(* PLC project Astro, Actility iec61131 1.0.28, author Laurent Nicq *)
(* stored: creationDateTime 2013-03-20T17:09:43, version 1.1.2, modificationDateTime 2013-07-26T10:44:38 *)

(* Example for using the Sunset *)
PROGRAM POU_Astro_Using
  VAR_EXTERNAL
    GL_Astro_Status : DINT;
    GL_Current_DateTime : DT;
    GL_SunSet_Time : DT;
  END_VAR
  VAR
    Information : STRING;
    astro_status : DINT := 0;
    delay_before : TIME := t#30s;
    time_remaining : TIME;  (* temporary for debug *)
    delay_after : TIME := t#45s;
    light : BOOL := FALSE;
    current_day : DINT;
  END_VAR

(* transition new_day *)
yday(GL_Current_DateTime)<> current_day;
/* check for a different day. Avoid dealing with 365-366 days case */
              
(* Need to wait for a new day before using a
SunSet value calculated by the Astro script *)
INITIAL_STEP Get_status:
  GET_STATUS_INLINE1(N);
END_STEP
ACTION GET_STATUS_INLINE1:
  astro_status:= GL_Astro_Status;
END_ACTION
TRANSITION FROM Get_status TO Display_Status
  := astro_status <>0;
END_TRANSITION
TRANSITION FROM Get_status TO Astro_OK
  := astro_status = 0;
END_TRANSITION
STEP Display_Status:
  DISPLAY_STATUS_INLINE2(P);
END_STEP
ACTION DISPLAY_STATUS_INLINE2:
  Information:='Astro is NOT RUNNING';
END_ACTION
TRANSITION FROM Display_Status TO Get_status
  := TRUE;
END_TRANSITION
STEP Astro_OK:
  ASTRO_OK_INLINE3(P);
  store_current_day(N);
  remaining(N);
END_STEP
ACTION ASTRO_OK_INLINE3:
  Information:='Astro is RUNNING';
END_ACTION
TRANSITION FROM Astro_OK TO Start_SunSet
  := GL_Current_DateTime > GL_SunSet_Time - delay_before;
END_TRANSITION
STEP Start_SunSet:
  START_SUNSET_INLINE4(P);
END_STEP
ACTION START_SUNSET_INLINE4:
  light:=TRUE;
END_ACTION
TRANSITION FROM Start_SunSet TO Stop_SunSet
  := GL_Current_DateTime > (( GL_SunSet_Time - delay_before) + delay_after);
END_TRANSITION
STEP Stop_SunSet:
  STOP_SUNSET_INLINE5(P);
END_STEP
ACTION STOP_SUNSET_INLINE5:
  light:=FALSE;
END_ACTION
TRANSITION FROM Stop_SunSet TO Get_status
  := new_day;
END_TRANSITION

ACTION store_current_day:
current_day:= yday(GL_Current_DateTime);
              
END_ACTION

ACTION remaining:
time_remaining:= SUB_DT_DT(GL_SunSet_Time , GL_Current_DateTime);
              
END_ACTION
END_PROGRAM

(* Distributes the Sunset Sunrise times *)
PROGRAM POU_Astro_Sun_Time
  VAR_EXTERNAL
    GL_SunSet_Time : DT;
    GL_SunRise_Time : DT;
    GL_Current_DateTime : DT;
    GL_Astro_Status : INT;
    GL_Lat : REAL;
    GL_Lon : REAL;
  END_VAR
  VAR
    Astro_Version : STRING := '1.1.2';
    current_day : DINT;
    Lat : REAL := 0;
    Lon : REAL := 0;
  END_VAR

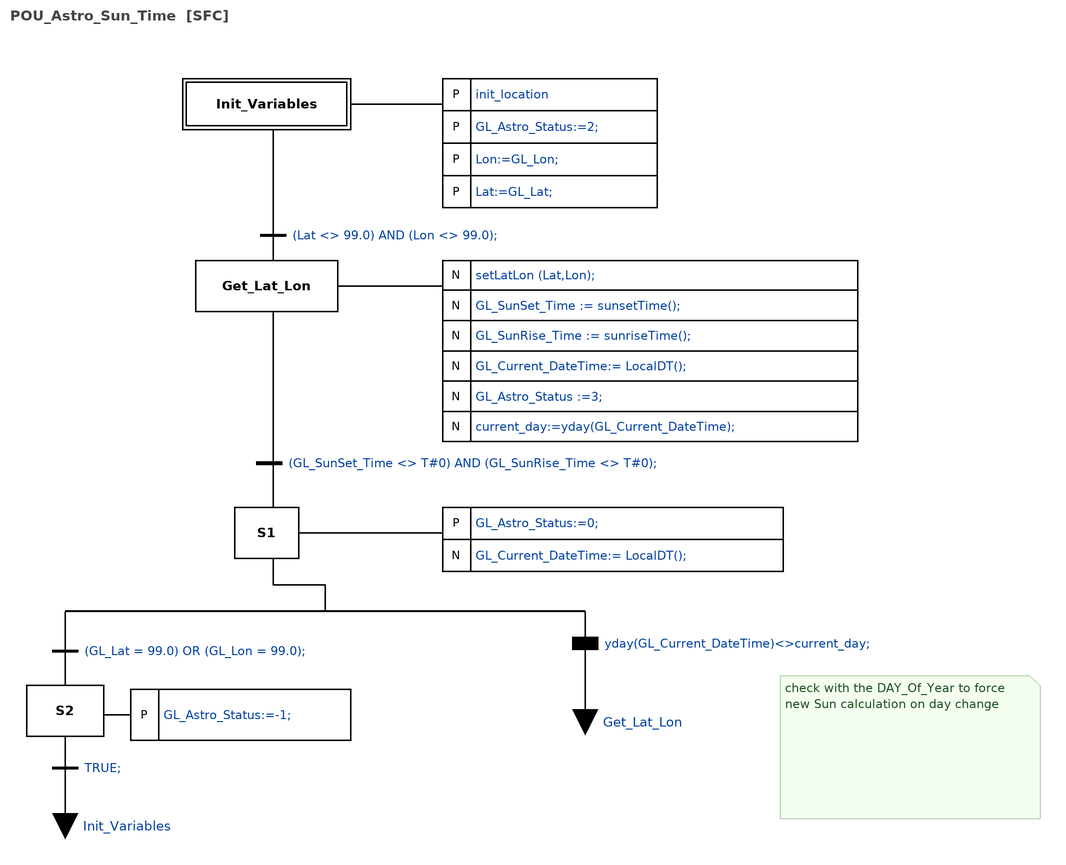
(* check with the DAY_Of_Year to force new Sun calculation on day change *)
INITIAL_STEP Init_Variables:
  init_location(P);
  INIT_VARIABLES_INLINE1(P);
  INIT_VARIABLES_INLINE2(P);
  INIT_VARIABLES_INLINE3(P);
END_STEP
ACTION INIT_VARIABLES_INLINE1:
  GL_Astro_Status:=2;
END_ACTION
ACTION INIT_VARIABLES_INLINE2:
  Lon:=GL_Lon;
END_ACTION
ACTION INIT_VARIABLES_INLINE3:
  Lat:=GL_Lat;
END_ACTION
TRANSITION FROM Init_Variables TO Get_Lat_Lon
  := (Lat <> 99.0) AND (Lon <> 99.0);
END_TRANSITION
STEP Get_Lat_Lon:
  GET_LAT_LON_INLINE4(N);
  GET_LAT_LON_INLINE5(N);
  GET_LAT_LON_INLINE6(N);
  GET_LAT_LON_INLINE7(N);
  GET_LAT_LON_INLINE8(N);
  GET_LAT_LON_INLINE9(N);
END_STEP
ACTION GET_LAT_LON_INLINE4:
  setLatLon (Lat,Lon);
END_ACTION
ACTION GET_LAT_LON_INLINE5:
  GL_SunSet_Time := sunsetTime();
END_ACTION
ACTION GET_LAT_LON_INLINE6:
  GL_SunRise_Time := sunriseTime();
END_ACTION
ACTION GET_LAT_LON_INLINE7:
  GL_Current_DateTime:= LocalDT();
END_ACTION
ACTION GET_LAT_LON_INLINE8:
  GL_Astro_Status :=3;
END_ACTION
ACTION GET_LAT_LON_INLINE9:
  current_day:=yday(GL_Current_DateTime);
END_ACTION
TRANSITION FROM Get_Lat_Lon TO S1
  := (GL_SunSet_Time <> T#0) AND (GL_SunRise_Time <> T#0);
END_TRANSITION
STEP S1:
  S1_INLINE10(P);
  S1_INLINE11(N);
END_STEP
ACTION S1_INLINE10:
  GL_Astro_Status:=0;
END_ACTION
ACTION S1_INLINE11:
  GL_Current_DateTime:= LocalDT();
END_ACTION
TRANSITION FROM S1 TO S2
  := (GL_Lat = 99.0) OR (GL_Lon = 99.0);
END_TRANSITION
TRANSITION FROM S1 TO Get_Lat_Lon
  := yday(GL_Current_DateTime)<>current_day;
END_TRANSITION
STEP S2:
  S2_INLINE12(P);
END_STEP
ACTION S2_INLINE12:
  GL_Astro_Status:=-1;
END_ACTION
TRANSITION FROM S2 TO Init_Variables
  := TRUE;
END_TRANSITION

ACTION init_location:
/* Lyon, France */
GL_Lat:=45.76404;
GL_Lon:=4.835659;
/* Narvik, Norway */
/* (no sunset in june and no sunrise in december) */
/* GL_Lat:=68.433; */
/* GL_Lon:=17.4167; */
              
END_ACTION
END_PROGRAM

CONFIGURATION Astro_test
  RESOURCE Resource_main ON PLC
    VAR_GLOBAL
      GL_SunSet_Time : DT := T#0;
      GL_SunRise_Time : DT := T#0;
      GL_Current_DateTime : DT;
      GL_Astro_Status : DINT := -1;  (* -1 means Stopped *)
      GL_Lat : REAL := -99.0;  (* -99.0 means not initialized *)
      GL_Lon : REAL := -99.0;  (* -99.0 means not initialized *)
    END_VAR
    TASK task_slow(INTERVAL := T#5s0ms, PRIORITY := 0);
    TASK task_fast(INTERVAL := T#1s0ms, PRIORITY := 0);
    PROGRAM Instance_Astro_calc WITH task_slow : POU_Astro_Sun_Time;
    PROGRAM Instance_Astro_use WITH task_fast : POU_Astro_Using;
  END_RESOURCE
END_CONFIGURATION
